(* PLC project PLC Garden Controller, CODESYS CODESYS V3.5 SP16, author Toni Kucic *)
(* stored: creationDateTime 2021-03-29T22:16:35.9497507, version 1.0, modificationDateTime 2021-03-29T21:41:22.9745241, organization TK Automation *)
(* Automated gardening at its best. This is a portfolio project that features a simulator and a controller of four gardens holding 25 flowers/plants each. Each garden has a watering platform system moved by servo motors. In this project the user can learn how to control servo motors, optimize instruction/path algorithms and generally learn how to program PLCs. *)

TYPE Flower_typ : STRUCT
  x : INT;  (* X position of the flower cell in the HMI *)
  y : INT;  (* Y position of the flower cell in the HMI *)
  alpha : BYTE := 255;  (* Alpha channel *)
  red : BYTE := 2;  (* Red color channel *)
  green : BYTE := 253;  (* Green color channel *)
  blue : BYTE := 0;  (* Blue color channel *)
  color : DWORD;  (* Color variable to be used in the graphics *)
  hum : REAL := 100;  (* Humidity of the flower cell *)
  alive : BOOL := TRUE;  (* Flower is alive *)
END_STRUCT;
END_TYPE

TYPE Platform_typ : STRUCT
  x : INT;  (* Position from starting point on X axis *)
  y : INT;  (* Position from starting point on Y axis *)
  OpenValveCmd : BOOL;  (* Opens the water container valve *)
END_STRUCT;
END_TYPE

TYPE HMI_Cmds_typ : STRUCT
  CtrlOn : BOOL := TRUE;  (* Control is activated *)
  UpCmd : BOOL;  (* Command for platform UP *)
  DownCmd : BOOL;  (* Command for platform DOWN *)
  LeftCmd : BOOL;  (* Command for platform LEFT *)
  RightCmd : BOOL;  (* Command for platform RIGHT *)
  LeftUpCmd : BOOL;  (* Command for platform LEFT AND UP *)
  RightUpCmd : BOOL;  (* Command for platform RIGHT AND UP *)
  LeftDownCmd : BOOL;  (* Command for platform LEFT AND DOWN *)
  RightDownCmd : BOOL;  (* Command for platform RIGHT AND DOWN *)
  OpenWaterValve : BOOL;  (* Command to open the water valve *)
END_STRUCT;
END_TYPE

FUNCTION BYTES_TO_DWORD : DWORD
  VAR_INPUT
    B0 : BYTE;  (* Least significant byte *)
    B1 : BYTE;  (* Byte two *)
    B2 : BYTE;  (* Byte three *)
    B3 : BYTE;  (* Highest significant byte *)
  END_VAR

            BYTES_TO_DWORD.0 := B0.0;
BYTES_TO_DWORD.1 := B0.1;
BYTES_TO_DWORD.2 := B0.2;
BYTES_TO_DWORD.3 := B0.3;
BYTES_TO_DWORD.4 := B0.4;
BYTES_TO_DWORD.5 := B0.5;
BYTES_TO_DWORD.6 := B0.6;
BYTES_TO_DWORD.7 := B0.7;

BYTES_TO_DWORD.8 := B1.0;
BYTES_TO_DWORD.9 := B1.1;
BYTES_TO_DWORD.10 := B1.2;
BYTES_TO_DWORD.11 := B1.3;
BYTES_TO_DWORD.12 := B1.4;
BYTES_TO_DWORD.13 := B1.5;
BYTES_TO_DWORD.14 := B1.6;
BYTES_TO_DWORD.15 := B1.7;

BYTES_TO_DWORD.16 := B2.0;
BYTES_TO_DWORD.17 := B2.1;
BYTES_TO_DWORD.18 := B2.2;
BYTES_TO_DWORD.19 := B2.3;
BYTES_TO_DWORD.20 := B2.4;
BYTES_TO_DWORD.21 := B2.5;
BYTES_TO_DWORD.22 := B2.6;
BYTES_TO_DWORD.23 := B2.7;

BYTES_TO_DWORD.24 := B3.0;
BYTES_TO_DWORD.25 := B3.1;
BYTES_TO_DWORD.26 := B3.2;
BYTES_TO_DWORD.27 := B3.3;
BYTES_TO_DWORD.28 := B3.4;
BYTES_TO_DWORD.29 := B3.5;
BYTES_TO_DWORD.30 := B3.6;
BYTES_TO_DWORD.31 := B3.7;
RETURN;
          
END_FUNCTION

FUNCTION_BLOCK ClockPulse
  VAR_INPUT
    f : TIME := TIME#500ms;  (* Oscillate once per f *)
  END_VAR
  VAR_OUTPUT
    pulse : BOOL;  (* Pulse for use. One cycle *)
  END_VAR
  VAR
    edge : R_TRIG;
    clock : BLINK;
  END_VAR

            clock(ENABLE:=TRUE, TIMELOW:=f, TIMEHIGH:=f);
edge(CLK:=clock.OUT);
pulse := edge.Q;
          
END_FUNCTION_BLOCK

FUNCTION checkOverlapRectangle : BOOL
  VAR_INPUT
    R1_X : INT;  (* Rectangle 1 x position *)
    R1_Y : INT;  (* Rectangle 1 y position *)
    R1_W : INT;  (* Rectangle 1 width *)
    R1_H : INT;  (* Rectangle 1 height *)
    R2_X : INT;  (* Rectangle 2 x position *)
    R2_Y : INT;  (* Rectangle 2 y position *)
    R2_W : INT;  (* Rectangle 2 width *)
    R2_H : INT;  (* Rectangle 2 height *)
  END_VAR

            (*Calculate if these two rectangles are overlapping*)
IF R1_X < (R2_X + R2_W) AND
   (R1_X + R1_W) > R2_X AND
   R1_Y < (R2_Y + R2_H) AND
  (R1_H + R1_Y) > R2_Y THEN
   checkOverlapRectangle := TRUE;
ELSE
	checkOverlapRectangle := FALSE;
END_IF
          
END_FUNCTION

PROGRAM simu
  VAR
    clock : ClockPulse;  (* Clock pulse for the program *)
    i : UINT;  (* Iterator variable *)
    vG1PlantsAlive : UINT;  (* Number of plants alive in garden 1 *)
    vG2PlantsAlive : UINT;  (* Number of plants alive in garden 2 *)
    vG3PlantsAlive : UINT;  (* Number of plants alive in garden 3 *)
    vG4PlantsAlive : UINT;  (* Number of plants alive in garden 4 *)
    vGarden1 : ARRAY[0..24] OF Flower_typ := [(x := 42, y := 42), (x := 122, y := 42), (x := 202, y := 42), (x := 282, y := 42), (x := 362, y := 42), (x := 42, y := 122), (x := 122, y := 122), (x := 202, y := 122), (x := 282, y := 122), (x := 362, y := 122), (x := 42, y := 202), (x := 122, y := 202), (x := 202, y := 202), (x := 282, y := 202), (x := 362, y := 202), (x := 42, y := 282), (x := 122, y := 282), (x := 202, y := 282), (x := 282, y := 282), (x := 362, y := 282), (x := 42, y := 362), (x := 122, y := 362), (x := 202, y := 362), (x := 282, y := 362), (x := 362, y := 362)];  (* Locations of plant cells in the HMI for the garden 1. Not to be mistaken with servo offset *)
    vGarden2 : ARRAY[0..24] OF Flower_typ := [(x := 642, y := 42), (x := 722, y := 42), (x := 802, y := 42), (x := 882, y := 42), (x := 962, y := 42), (x := 642, y := 122), (x := 722, y := 122), (x := 802, y := 122), (x := 882, y := 122), (x := 962, y := 122), (x := 642, y := 202), (x := 722, y := 202), (x := 802, y := 202), (x := 882, y := 202), (x := 962, y := 202), (x := 642, y := 282), (x := 722, y := 282), (x := 802, y := 282), (x := 882, y := 282), (x := 962, y := 282), (x := 642, y := 362), (x := 722, y := 362), (x := 802, y := 362), (x := 882, y := 362), (x := 962, y := 362)];  (* Locations of plant cells in the HMI for the garden 2. Not to be mistaken with servo offset *)
    vGarden3 : ARRAY[0..24] OF Flower_typ := [(x := 42, y := 642), (x := 122, y := 642), (x := 202, y := 642), (x := 282, y := 642), (x := 362, y := 642), (x := 42, y := 722), (x := 122, y := 722), (x := 202, y := 722), (x := 282, y := 722), (x := 362, y := 722), (x := 42, y := 802), (x := 122, y := 802), (x := 202, y := 802), (x := 282, y := 802), (x := 362, y := 802), (x := 42, y := 882), (x := 122, y := 882), (x := 202, y := 882), (x := 282, y := 882), (x := 362, y := 882), (x := 42, y := 962), (x := 122, y := 962), (x := 202, y := 962), (x := 282, y := 962), (x := 362, y := 962)];  (* Locations of plant cells in the HMI for the garden 3. Not to be mistaken with servo offset *)
    vGarden4 : ARRAY[0..24] OF Flower_typ := [(x := 642, y := 642), (x := 722, y := 642), (x := 802, y := 642), (x := 882, y := 642), (x := 962, y := 642), (x := 642, y := 722), (x := 722, y := 722), (x := 802, y := 722), (x := 882, y := 722), (x := 962, y := 722), (x := 642, y := 802), (x := 722, y := 802), (x := 802, y := 802), (x := 882, y := 802), (x := 962, y := 802), (x := 642, y := 882), (x := 722, y := 882), (x := 802, y := 882), (x := 882, y := 882), (x := 962, y := 882), (x := 642, y := 962), (x := 722, y := 962), (x := 802, y := 962), (x := 882, y := 962), (x := 962, y := 962)];  (* Locations of plant cells in the HMI for the garden 4. Not to be mistaken with servo offset *)
    vGarden1Platform : Platform_typ;  (* Platform 1 properties like x,y, water valve open etc *)
    vGarden2Platform : Platform_typ;  (* Platform 2 properties like x,y, water valve open etc *)
    vGarden3Platform : Platform_typ;  (* Platform 3 properties like x,y, water valve open etc *)
    vGarden4Platform : Platform_typ;  (* Platform 4 properties like x,y, water valve open etc *)
  END_VAR

                    (* SIMULATOR FUNCTIONAL DESCRIPTION
FLOWERS SIMULATION:
- there are 25 flowers in each garden
- each flower consumes humidity for life, this is represented as a number, this draw is constant
- each flower, if it has no humidity, it start decaying, decaying is represented with color
if color is red, the flower dies, if its green or yellow it is still alive
- if the flower gets too much water (>200%) this has same effect as it being too dry so the 
platform controller must maintain a proper level of humidity.
- there are no humidity sensors deployed to the gIO structure but if the user wants to, it is very easy

PLATFORM SIMULATION:
- platforms consist out of one Y Axis servo and two X axis servos
- X axis servos are electrically connected so they move as one for simplicity
- each servo motor is reporting its offset from the beggining of the servo
- for simplicity, each servo starts at 0 offset. If necessary, these starting points can be initialized
- commands CW increase the axis while CCW decrease the axis
- servo motors are identical but they are  flipped horizontally or verticaly, depending on the garden
but they always follow CW and CCW commands respectively
- upon command the open water valve releases the onboard stored water. For simplicity, the platform has 
unlimited supply of water

PLATFORM/FLOWER INTERACTION SIMULATION:
- if the nozzle (not the whole platform) of the platform is above a flower cell (80x80 pixels)
and the water valve is open, the flowers humidity increases
- the flower cells are divided by 1 px width and the nozzle is 10px wide so it is possible to
water multiple cells at once

COUNTING OF ALIVE FLOWERS:
- for each garden a counting of alive plants is done and it is displayed in the HMI*)

clock(f:=T#20MS);

(*Run the garden simulators*)
SIMULATE_GARDEN1();
SIMULATE_GARDEN2();
SIMULATE_GARDEN3();
SIMULATE_GARDEN4();
                  

ACTION SIMULATE_GARDEN1:
                        (*COLOR : 16# XX XX XX XX*)
(*            A  R  G  B *)
vG1PlantsAlive := 0;
FOR i:=0 TO 24 DO
	(*Simulate the humidity of one flower cell*)
	(*If not being watered, it slowly looses humidity*)
	vGarden1[i].hum := MAX(0, vGarden1[i].hum - 0.07 * BOOL_TO_REAL(clock.pulse));
	
	(*If the watering platform is above the cell, water valve is open and tank has water, increase the humidity*)
	IF checkOverlapRectangle(R1_X:=vGarden1[i].x, R1_Y:=vGarden1[i].y, R1_W:=80, R1_H:=80,
							R2_X:=406 + vGarden1Platform.x + 45, R2_Y:=361 + vGarden1Platform.y + 45, R2_W:=10, R2_H:=10) AND vGarden1Platform.OpenValveCmd THEN
		vGarden1[i].hum := vGarden1[i].hum + 4 * BOOL_TO_REAL(clock.pulse);
	END_IF
	
	(*Simulate flowers response to the humidity of the cell*)
	(*Flag if the plant is alive*)
	vGarden1[i].alive := NOT (vGarden1[i].red >= 254 AND vGarden1[i].green < 100);
	IF vGarden1[i].hum <= 0 OR vGarden1[i].hum >= 200 THEN
		(*Flower starts decaying if not enough or too much humiditiy*)
		(*Change color towards red*)
		vGarden1[i].red := vGarden1[i].red + 1 * BOOL_TO_BYTE(clock.pulse);
		vGarden1[i].green := vGarden1[i].green - 1 * BOOL_TO_BYTE(clock.pulse AND vGarden1[i].red > 253);
	ELSE
		IF vGarden1[i].alive THEN
			(*Flower gets better much faster than it dies*)
			(*Change color towards green*)
			vGarden1[i].green := vGarden1[i].green + 1 * BOOL_TO_BYTE(clock.pulse);
			vGarden1[i].red := vGarden1[i].red - 1 * BOOL_TO_BYTE(clock.pulse AND vGarden1[i].green > 253);
		(*ELSE It is dead for good*)
			
		END_IF
	END_IF
	vGarden1[i].red := LIMIT(1, vGarden1[i].red, 254);
	vGarden1[i].green := LIMIT(1, vGarden1[i].green, 254);
	
	(*Combine the channel bytes into dword color*)
	vGarden1[i].color := BYTES_TO_DWORD(B0 := vGarden1[i].blue,B1 := vGarden1[i].green,
										B2 := vGarden1[i].red, B3 := vGarden1[i].alpha);
										
	(*Count how many plants are alive*)
	vG1PlantsAlive := vG1PlantsAlive + BOOL_TO_UINT(vGarden1[i].alive);
END_FOR

(*Servo motors*)
(*Move on X*)
IF gIO.Garden1_ServoX_CCW THEN
	vGarden1Platform.x := vGarden1Platform.x + 1;
ELSIF gIO.Garden1_ServoX_CW THEN
	vGarden1Platform.x := vGarden1Platform.x - 1;
END_IF
(*Limit the platforms movement on x axis*)
vGarden1Platform.x := LIMIT(-404, vGarden1Platform.x, 0);
(*Move on Y*)
IF gIO.Garden1_ServoY_CCW THEN
	vGarden1Platform.y := vGarden1Platform.y + 1;
ELSIF gIO.Garden1_ServoY_CW THEN
	vGarden1Platform.y := vGarden1Platform.y - 1;
END_IF
(*Limit the platforms movement on y axis*)
vGarden1Platform.y := LIMIT(-320, vGarden1Platform.y, 0);

(*Report the position of the platform*)
gIO.Garden1_ServoX_Offset := ABS(vGarden1Platform.x);
gIO.Garden1_ServoY_Offset := ABS(vGarden1Platform.y);

(*Control the water valve*)
vGarden1Platform.OpenValveCmd := gIO.Garden1_WaterTankOpenCmd;
                      
END_ACTION

ACTION SIMULATE_GARDEN2:
                        (*COLOR : 16# XX XX XX XX*)
(*            A  R  G  B *)
vG2PlantsAlive := 0;
FOR i:=0 TO 24 DO
	(*Simulate the humidity of one flower cell*)
	(*If not being watered, it slowly looses humidity*)
	vGarden2[i].hum := MAX(0, vGarden2[i].hum - 0.07 * BOOL_TO_REAL(clock.pulse));
	
	(*If the watering platform is above the cell, water valve is open and tank has water, increase the humidity*)
	IF checkOverlapRectangle(R1_X:=vGarden2[i].x, R1_Y:=vGarden2[i].y, R1_W:=80, R1_H:=80,
							R2_X:=594 + vGarden2Platform.x + 45, R2_Y:=361 + vGarden2Platform.y + 45, R2_W:=10, R2_H:=10) AND vGarden2Platform.OpenValveCmd THEN
		vGarden2[i].hum := vGarden2[i].hum + 4 * BOOL_TO_REAL(clock.pulse);
	END_IF
	
	(*Simulate flowers response to the humidity of the cell*)
	(*Flag if the plant is alive*)
	vGarden2[i].alive := NOT (vGarden2[i].red >= 254 AND vGarden2[i].green < 100);
	IF vGarden2[i].hum <= 0 OR vGarden2[i].hum >= 200 THEN
		(*Flower starts decaying if not enough or too much humiditiy*)
		(*Change color towards red*)
		vGarden2[i].red := vGarden2[i].red + 1 * BOOL_TO_BYTE(clock.pulse);
		vGarden2[i].green := vGarden2[i].green - 1 * BOOL_TO_BYTE(clock.pulse AND vGarden2[i].red > 253);
	ELSE
		IF vGarden2[i].alive THEN
			(*Flower gets better much faster than it dies*)
			(*Change color towards green*)
			vGarden2[i].green := vGarden2[i].green + 1 * BOOL_TO_BYTE(clock.pulse);
			vGarden2[i].red := vGarden2[i].red - 1 * BOOL_TO_BYTE(clock.pulse AND vGarden2[i].green > 253);
		(*ELSE It is dead for good*)
			
		END_IF
	END_IF
	vGarden2[i].red := LIMIT(1, vGarden2[i].red, 254);
	vGarden2[i].green := LIMIT(1, vGarden2[i].green, 254);
	
	(*Combine the channel bytes into dword color*)
	vGarden2[i].color := BYTES_TO_DWORD(B0 := vGarden2[i].blue,B1 := vGarden2[i].green,
										B2 := vGarden2[i].red, B3 := vGarden2[i].alpha);
										
	(*Count how many plants are alive*)
	vG2PlantsAlive := vG2PlantsAlive + BOOL_TO_UINT(vGarden2[i].alive);
END_FOR

(*Servo motors*)
(*Move on X*)
IF gIO.Garden2_ServoX_CCW THEN
	vGarden2Platform.x := vGarden2Platform.x - 1;
ELSIF gIO.Garden2_ServoX_CW THEN
	vGarden2Platform.x := vGarden2Platform.x + 1;
END_IF
(*Limit the platforms movement on x axis*)
vGarden2Platform.x := LIMIT(0, vGarden2Platform.x, 404);
(*Move on Y*)
IF gIO.Garden2_ServoY_CCW THEN
	vGarden2Platform.y := vGarden2Platform.y + 1;
ELSIF gIO.Garden2_ServoY_CW THEN
	vGarden2Platform.y := vGarden2Platform.y - 1;
END_IF
(*Limit the platforms movement on y axis*)
vGarden2Platform.y := LIMIT(-320, vGarden2Platform.y, 0);

(*Report the position of the platform*)
gIO.Garden2_ServoX_Offset := ABS(vGarden2Platform.x);
gIO.Garden2_ServoY_Offset := ABS(vGarden2Platform.y);

(*Control the water valve*)
vGarden2Platform.OpenValveCmd := gIO.Garden2_WaterTankOpenCmd;
                      
END_ACTION

ACTION SIMULATE_GARDEN3:
                        (*COLOR : 16# XX XX XX XX*)
(*            A  R  G  B *)
vG3PlantsAlive := 0;
FOR i:=0 TO 24 DO
	(*Simulate the humidity of one flower cell*)
	(*If not being watered, it slowly looses humidity*)
	vGarden3[i].hum := MAX(0, vGarden3[i].hum - 0.07 * BOOL_TO_REAL(clock.pulse));
	
	(*If the watering platform is above the cell, water valve is open and tank has water, increase the humidity*)
	IF checkOverlapRectangle(R1_X:=vGarden3[i].x, R1_Y:=vGarden3[i].y, R1_W:=80, R1_H:=80,
							R2_X:=401 + vGarden3Platform.x + 45, R2_Y:=640 + vGarden3Platform.y + 45, R2_W:=10, R2_H:=10) AND vGarden3Platform.OpenValveCmd THEN
		vGarden3[i].hum := vGarden3[i].hum + 4 * BOOL_TO_REAL(clock.pulse);
	END_IF
	
	(*Simulate flowers response to the humidity of the cell*)
	(*Flag if the plant is alive*)
	vGarden3[i].alive := NOT (vGarden3[i].red >= 254 AND vGarden3[i].green < 100);
	IF vGarden3[i].hum <= 0 OR vGarden3[i].hum >= 200 THEN
		(*Flower starts decaying if not enough or too much humiditiy*)
		(*Change color towards red*)
		vGarden3[i].red := vGarden3[i].red + 1 * BOOL_TO_BYTE(clock.pulse);
		vGarden3[i].green := vGarden3[i].green - 1 * BOOL_TO_BYTE(clock.pulse AND vGarden3[i].red > 253);
	ELSE
		IF vGarden3[i].alive THEN
			(*Flower gets better much faster than it dies*)
			(*Change color towards green*)
			vGarden3[i].green := vGarden3[i].green + 1 * BOOL_TO_BYTE(clock.pulse);
			vGarden3[i].red := vGarden3[i].red - 1 * BOOL_TO_BYTE(clock.pulse AND vGarden3[i].green > 253);
		(*ELSE It is dead for good*)
			
		END_IF
	END_IF
	vGarden3[i].red := LIMIT(1, vGarden3[i].red, 254);
	vGarden3[i].green := LIMIT(1, vGarden3[i].green, 254);
	
	(*Combine the channel bytes into dword color*)
	vGarden3[i].color := BYTES_TO_DWORD(B0 := vGarden3[i].blue,B1 := vGarden3[i].green,
										B2 := vGarden3[i].red, B3 := vGarden3[i].alpha);
										
	(*Count how many plants are alive*)
	vG3PlantsAlive := vG3PlantsAlive + BOOL_TO_UINT(vGarden3[i].alive);
END_FOR

(*Servo motors*)
(*Move on X*)
IF gIO.Garden3_ServoX_CCW THEN
	vGarden3Platform.x := vGarden3Platform.x + 1;
ELSIF gIO.Garden3_ServoX_CW THEN
	vGarden3Platform.x := vGarden3Platform.x - 1;
END_IF
(*Limit the platforms movement on x axis*)
vGarden3Platform.x := LIMIT(-404, vGarden3Platform.x, 0);
(*Move on Y*)
IF gIO.Garden3_ServoY_CCW THEN
	vGarden3Platform.y := vGarden3Platform.y - 1;
ELSIF gIO.Garden3_ServoY_CW THEN
	vGarden3Platform.y := vGarden3Platform.y + 1;
END_IF
(*Limit the platforms movement on y axis*)
vGarden3Platform.y := LIMIT(0, vGarden3Platform.y, 320);

(*Report the position of the platform*)
gIO.Garden3_ServoX_Offset := ABS(vGarden3Platform.x);
gIO.Garden3_ServoY_Offset := ABS(vGarden3Platform.y);

(*Control the water valve*)
vGarden3Platform.OpenValveCmd := gIO.Garden3_WaterTankOpenCmd;
                      
END_ACTION

ACTION SIMULATE_GARDEN4:
                        (*COLOR : 16# XX XX XX XX*)
(*            A  R  G  B *)
vG4PlantsAlive := 0;
FOR i:=0 TO 24 DO
	(*Simulate the humidity of one flower cell*)
	(*If not being watered, it slowly looses humidity*)
	vGarden4[i].hum := MAX(0, vGarden4[i].hum - 0.07 * BOOL_TO_REAL(clock.pulse));
	
	(*If the watering platform is above the cell, water valve is open and tank has water, increase the humidity*)
	IF checkOverlapRectangle(R1_X:=vGarden4[i].x, R1_Y:=vGarden4[i].y, R1_W:=80, R1_H:=80,
							R2_X:=600 + vGarden4Platform.x + 45, R2_Y:=642 + vGarden4Platform.y + 45, R2_W:=10, R2_H:=10) AND vGarden4Platform.OpenValveCmd THEN
		vGarden4[i].hum := vGarden4[i].hum + 4 * BOOL_TO_REAL(clock.pulse);
	END_IF
	
	(*Simulate flowers response to the humidity of the cell*)
	(*Flag if the plant is alive*)
	vGarden4[i].alive := NOT (vGarden4[i].red >= 254 AND vGarden4[i].green < 100);
	IF vGarden4[i].hum <= 0 OR vGarden4[i].hum >= 200 THEN
		(*Flower starts decaying if not enough or too much humiditiy*)
		(*Change color towards red*)
		vGarden4[i].red := vGarden4[i].red + 1 * BOOL_TO_BYTE(clock.pulse);
		vGarden4[i].green := vGarden4[i].green - 1 * BOOL_TO_BYTE(clock.pulse AND vGarden4[i].red > 253);
	ELSE
		IF vGarden4[i].alive THEN
			(*Flower gets better much faster than it dies*)
			(*Change color towards green*)
			vGarden4[i].green := vGarden4[i].green + 1 * BOOL_TO_BYTE(clock.pulse);
			vGarden4[i].red := vGarden4[i].red - 1 * BOOL_TO_BYTE(clock.pulse AND vGarden4[i].green > 253);
		(*ELSE It is dead for good*)
			
		END_IF
	END_IF
	vGarden4[i].red := LIMIT(1, vGarden4[i].red, 254);
	vGarden4[i].green := LIMIT(1, vGarden4[i].green, 254);
	
	(*Combine the channel bytes into dword color*)
	vGarden4[i].color := BYTES_TO_DWORD(B0 := vGarden4[i].blue,B1 := vGarden4[i].green,
										B2 := vGarden4[i].red, B3 := vGarden4[i].alpha);
										
	(*Count how many plants are alive*)
	vG4PlantsAlive := vG4PlantsAlive + BOOL_TO_UINT(vGarden4[i].alive);
END_FOR

(*Servo motors*)
(*Move on X*)
IF gIO.Garden4_ServoX_CCW THEN
	vGarden4Platform.x := vGarden4Platform.x - 1;
ELSIF gIO.Garden4_ServoX_CW THEN
	vGarden4Platform.x := vGarden4Platform.x + 1;
END_IF
(*Limit the platforms movement on x axis*)
vGarden4Platform.x := LIMIT(0, vGarden4Platform.x, 404);
(*Move on Y*)
IF gIO.Garden4_ServoY_CCW THEN
	vGarden4Platform.y := vGarden4Platform.y - 1;
ELSIF gIO.Garden4_ServoY_CW THEN
	vGarden4Platform.y := vGarden4Platform.y + 1;
END_IF
(*Limit the platforms movement on y axis*)
vGarden4Platform.y := LIMIT(0, vGarden4Platform.y, 320);

(*Report the position of the platform*)
gIO.Garden4_ServoX_Offset := ABS(vGarden4Platform.x);
gIO.Garden4_ServoY_Offset := ABS(vGarden4Platform.y);

(*Control the water valve*)
vGarden4Platform.OpenValveCmd := gIO.Garden4_WaterTankOpenCmd;
                      
END_ACTION
END_PROGRAM

PROGRAM main
  VAR
    vG1Platform_Instructions : ARRAY[0..24, 0..1] OF INT := [365, 320, 285, 320, 205, 320, 125, 320, 45, 320, 45, 240, 125, 240, 205, 240, 285, 240, 365, 240, 365, 160, 285, 160, 205, 160, 125, 160, 45, 160, 45, 80, 125, 80, 205, 80, 285, 80, 365, 80, 365, 0, 285, 0, 205, 0, 125, 0, 45, 0];  (* Instructions for platform servos in garden 1 *)
    vG2Platform_Instructions : ARRAY[0..24, 0..1] OF INT := [50, 320, 50, 240, 50, 160, 50, 80, 50, 0, 130, 0, 130, 80, 130, 160, 130, 240, 130, 320, 210, 320, 210, 240, 210, 160, 210, 80, 210, 0, 290, 0, 290, 80, 290, 160, 290, 240, 290, 320, 370, 320, 370, 240, 370, 160, 370, 80, 370, 0];  (* Instructions for platform servos in garden 2 *)
    vG3Platform_Instructions : ARRAY[0..24, 0..1] OF INT := [358, 0, 278, 0, 358, 80, 358, 160, 278, 80, 198, 0, 118, 0, 198, 80, 278, 160, 358, 240, 358, 320, 278, 240, 198, 160, 118, 80, 38, 0, 38, 80, 118, 160, 198, 240, 278, 320, 198, 320, 118, 240, 38, 160, 38, 240, 118, 320, 38, 320];  (* Instructions for platform servos in garden 3 *)
    vG4Platform_Instructions : ARRAY[0..24, 0..1] OF INT := [200, 160, 120, 160, 120, 240, 200, 240, 280, 240, 280, 160, 280, 80, 200, 80, 120, 80, 40, 80, 40, 160, 40, 240, 40, 320, 120, 320, 200, 320, 280, 320, 360, 320, 360, 240, 360, 160, 360, 80, 360, 0, 280, 0, 200, 0, 120, 0, 40, 0];  (* Instructions for platform servos in garden 4 *)
    garden1AutoWater : AutomaticFlowerWatering;  (* Automatic watering logic: Left to right in a smart way *)
    garden2AutoWater : AutomaticFlowerWatering;  (* Automatic watering logic: Going top to bottom in a smart way *)
    garden3AutoWater : AutomaticFlowerWatering;  (* Automatic watering logic: Going side ways from the top to bottom *)
    garden4AutoWater : AutomaticFlowerWatering;  (* Automatic watering logic: Goign from the middle out *)
  END_VAR

                    (*FUNCTIONAL DESCRIPTION:
- there are four gardens holding 25 flowers each
- the flowers need to be watered on a regular basis in order to keep their humidity in correct levels
- correct humidity is 0 > x < 200 %, if the humidity is not in those limits, the flower starts dying
- the watering is done by means of a watering platform, moved by x a y servos
- the job of this program is to move the platform of each garden and water the plants in an optimized way
- program should strive to keep all plants alive (easier said than done)
- the platforms move quite slowly as the water tank might spill so it is a given that 25 flower can be 
watered in 25 seconds
- on top of each platform there is a water tank with a valve that can be open remotely by the main program
- the program also needs to implement manual control from the HMI with the prepared variables in gIO structure
*)
CONTROL_GARDEN1();
CONTROL_GARDEN2();
CONTROL_GARDEN3();
CONTROL_GARDEN4();

                  

ACTION CONTROL_GARDEN1:
                        IF gIO.Garden1_HMI.CtrlOn THEN
	(*HMI Control*)
	gIO.Garden1_ServoX_CW := gIO.Garden1_HMI.LeftCmd OR gIO.Garden1_HMI.LeftDownCmd OR gIO.Garden1_HMI.LeftUpCmd;
	gIO.Garden1_ServoX_CCW := gIO.Garden1_HMI.RightCmd OR gIO.Garden1_HMI.RightDownCmd OR gIO.Garden1_HMI.RightUpCmd;
	
	gIO.Garden1_ServoY_CW := gIO.Garden1_HMI.UpCmd OR gIO.Garden1_HMI.LeftUpCmd OR gIO.Garden1_HMI.RightUpCmd;
	gIO.Garden1_ServoY_CCW := gIO.Garden1_HMI.DownCmd OR gIO.Garden1_HMI.LeftDownCmd OR gIO.Garden1_HMI.RightDownCmd;
	
	gIO.Garden1_WaterTankOpenCmd := gIO.Garden1_HMI.OpenWaterValve;
ELSE
	(*Automatic control*)
	garden1AutoWater(instructions:=vG1Platform_Instructions,
		xAxis := gIO.Garden1_ServoX_Offset,
		yAxis := gIO.Garden1_ServoY_Offset,
		servoX_CW => gIO.Garden1_ServoX_CW,
		servoX_CCW => gIO.Garden1_ServoX_CCW,
		servoY_CW => gIO.Garden1_ServoY_CW,
		servoY_CCW => gIO.Garden1_ServoY_CCW,
		waterTankOpenCmd => gIO.Garden1_WaterTankOpenCmd);
END_IF
                      
END_ACTION

ACTION CONTROL_GARDEN2:
                        IF gIO.Garden2_HMI.CtrlOn THEN
	(*HMI Control*)
	(*X servos are flipped on this garden*)
	gIO.Garden2_ServoX_CCW := gIO.Garden2_HMI.LeftCmd OR gIO.Garden2_HMI.LeftDownCmd OR gIO.Garden2_HMI.LeftUpCmd;
	gIO.Garden2_ServoX_CW := gIO.Garden2_HMI.RightCmd OR gIO.Garden2_HMI.RightDownCmd OR gIO.Garden2_HMI.RightUpCmd;
	
	gIO.Garden2_ServoY_CW := gIO.Garden2_HMI.UpCmd OR gIO.Garden2_HMI.LeftUpCmd OR gIO.Garden2_HMI.RightUpCmd;
	gIO.Garden2_ServoY_CCW := gIO.Garden2_HMI.DownCmd OR gIO.Garden2_HMI.LeftDownCmd OR gIO.Garden2_HMI.RightDownCmd;
	
	gIO.Garden2_WaterTankOpenCmd := gIO.Garden2_HMI.OpenWaterValve;
ELSE
	(*Automatic control*)
	garden2AutoWater(instructions:=vG2Platform_Instructions,
		xAxis := gIO.Garden2_ServoX_Offset,
		yAxis := gIO.Garden2_ServoY_Offset,
		servoX_CW => gIO.Garden2_ServoX_CW,
		servoX_CCW => gIO.Garden2_ServoX_CCW,
		servoY_CW => gIO.Garden2_ServoY_CW,
		servoY_CCW => gIO.Garden2_ServoY_CCW,
		waterTankOpenCmd => gIO.Garden2_WaterTankOpenCmd);
END_IF
                      
END_ACTION

ACTION CONTROL_GARDEN3:
                        IF gIO.Garden3_HMI.CtrlOn THEN
	(*HMI Control*)
	gIO.Garden3_ServoX_CW := gIO.Garden3_HMI.LeftCmd OR gIO.Garden3_HMI.LeftDownCmd OR gIO.Garden3_HMI.LeftUpCmd;
	gIO.Garden3_ServoX_CCW := gIO.Garden3_HMI.RightCmd OR gIO.Garden3_HMI.RightDownCmd OR gIO.Garden3_HMI.RightUpCmd;
	
	gIO.Garden3_ServoY_CCW := gIO.Garden3_HMI.UpCmd OR gIO.Garden3_HMI.LeftUpCmd OR gIO.Garden3_HMI.RightUpCmd;
	gIO.Garden3_ServoY_CW := gIO.Garden3_HMI.DownCmd OR gIO.Garden3_HMI.LeftDownCmd OR gIO.Garden3_HMI.RightDownCmd;
	
	gIO.Garden3_WaterTankOpenCmd := gIO.Garden3_HMI.OpenWaterValve;
ELSE
	(*Automatic control*)
	garden3AutoWater(instructions:=vG3Platform_Instructions,
		xAxis := gIO.Garden3_ServoX_Offset,
		yAxis := gIO.Garden3_ServoY_Offset,
		servoX_CW => gIO.Garden3_ServoX_CW,
		servoX_CCW => gIO.Garden3_ServoX_CCW,
		servoY_CW => gIO.Garden3_ServoY_CW,
		servoY_CCW => gIO.Garden3_ServoY_CCW,
		waterTankOpenCmd => gIO.Garden3_WaterTankOpenCmd);
END_IF
                      
END_ACTION

ACTION CONTROL_GARDEN4:
                        IF gIO.Garden4_HMI.CtrlOn THEN
	(*HMI Control*)
	gIO.Garden4_ServoX_CCW := gIO.Garden4_HMI.LeftCmd OR gIO.Garden4_HMI.LeftDownCmd OR gIO.Garden4_HMI.LeftUpCmd;
	gIO.Garden4_ServoX_CW := gIO.Garden4_HMI.RightCmd OR gIO.Garden4_HMI.RightDownCmd OR gIO.Garden4_HMI.RightUpCmd;
	
	gIO.Garden4_ServoY_CCW := gIO.Garden4_HMI.UpCmd OR gIO.Garden4_HMI.LeftUpCmd OR gIO.Garden4_HMI.RightUpCmd;
	gIO.Garden4_ServoY_CW := gIO.Garden4_HMI.DownCmd OR gIO.Garden4_HMI.LeftDownCmd OR gIO.Garden4_HMI.RightDownCmd;
	
	gIO.Garden4_WaterTankOpenCmd := gIO.Garden4_HMI.OpenWaterValve;
ELSE
	(*Automatic control*)
	garden4AutoWater(instructions:=vG4Platform_Instructions,
		xAxis := gIO.Garden4_ServoX_Offset,
		yAxis := gIO.Garden4_ServoY_Offset,
		servoX_CW => gIO.Garden4_ServoX_CW,
		servoX_CCW => gIO.Garden4_ServoX_CCW,
		servoY_CW => gIO.Garden4_ServoY_CW,
		servoY_CCW => gIO.Garden4_ServoY_CCW,
		waterTankOpenCmd => gIO.Garden4_WaterTankOpenCmd);
END_IF
                      
END_ACTION
END_PROGRAM

FUNCTION_BLOCK AutomaticFlowerWatering
  VAR_INPUT
    instructions : ARRAY[0..24, 0..1] OF INT;  (* Instructions to follow *)
    xAxis : INT;  (* Actual position of the X axis servo *)
    yAxis : INT;  (* Actual position of the Y axis servo *)
  END_VAR
  VAR_OUTPUT
    servoX_CW : BOOL;  (* Command to turn X axis servo clock wise *)
    servoX_CCW : BOOL;  (* Command to turn X axis servo counter clock wise *)
    servoY_CW : BOOL;  (* Command to turn Y axis servo clock wise *)
    servoY_CCW : BOOL;  (* Command to turn Y axis servo counter clock wise *)
    waterTankOpenCmd : BOOL;  (* Command to the platform to open the water valve *)
  END_VAR
  VAR
    i : UINT;  (* Iterator variable *)
    vXAxisCmd : INT;  (* Next X axis target *)
    vYAxisCmd : INT;  (* Next Y axis target *)
    vPlatformAtTarget : BOOL;  (* Flag for reaching the target *)
    WateringTimer : TON;  (* Timer for controlling the valve being open *)
  END_VAR

                    (* Parse the instruction to get new x and y targets *)
vXAxisCmd := instructions[i,0];
vYAxisCmd := instructions[i,1];
	
(*Check if the platform is at the target*)
vPlatformAtTarget := xAxis = vXAxisCmd AND yAxis = vYAxisCmd;

IF vPlatformAtTarget THEN
	(*Start watering for 1 second*)
	WateringTimer(IN:=TRUE, PT:=T#1S);
	waterTankOpenCmd := TRUE;
	
	(*If watering is finished, close valve and go to next flower*)
	IF WateringTimer.Q THEN
		WateringTimer(IN := FALSE);
		waterTankOpenCmd:= FALSE;
		i:= i + 1;
	END_IF
END_IF

(*If we traversed all instructions, go to first instruction*)
IF i = 25 THEN
	i := 0;
END_IF

(* Actual motor movement algorithm *)
IF vXAxisCmd > xAxis THEN
	servoX_CCW := FALSE;
	servoX_CW := TRUE;
ELSIF vXAxisCmd < xAxis THEN
	servoX_CCW := TRUE;
	servoX_CW := FALSE;
ELSE
	servoX_CCW := FALSE;
	servoX_CW := FALSE;
END_IF
	
IF vYAxisCmd < yAxis THEN
	servoY_CCW := TRUE;
	servoY_CW := FALSE;
ELSIF vYAxisCmd > yAxis THEN
	servoY_CCW := FALSE;
	servoY_CW := TRUE;
ELSE
	servoY_CCW := FALSE;
	servoY_CW := FALSE;
END_IF

	
                  
END_FUNCTION_BLOCK

CONFIGURATION SoftPLC
  RESOURCE Application ON PLC
    {attribute 'qualified_only'}
    VAR_GLOBAL  (* gIO *)
      Garden1_ServoX_CW : BOOL;  (* DO: Garden 1 servo X clock wise turn command *)
      Garden1_ServoX_CCW : BOOL;  (* DO: Garden 1 servo X counter clock wise turn command *)
      Garden1_ServoY_CW : BOOL;  (* DO: Garden 1 servo Y clock wise turn command *)
      Garden1_ServoY_CCW : BOOL;  (* DO: Garden 1 servo Y counter clock wise turn command *)
      Garden1_WaterTankOpenCmd : BOOL;  (* DO: Garden 1 water valve open command *)
      Garden2_ServoX_CW : BOOL;  (* DO: Garden 2 servo X clock wise turn command *)
      Garden2_ServoX_CCW : BOOL;  (* DO: Garden 2 servo X counter clock wise turn command *)
      Garden2_ServoY_CW : BOOL;  (* DO: Garden 2 servo Y clock wise turn command *)
      Garden2_ServoY_CCW : BOOL;  (* DO: Garden 2 servo Y counter clock wise turn command *)
      Garden2_WaterTankOpenCmd : BOOL;  (* DO: Garden 2 water valve open command *)
      Garden3_ServoX_CW : BOOL;  (* DO: Garden 3 servo X clock wise turn command *)
      Garden3_ServoX_CCW : BOOL;  (* DO: Garden 3 servo X counter clock wise turn command *)
      Garden3_ServoY_CW : BOOL;  (* DO: Garden 3 servo Y clock wise turn command *)
      Garden3_ServoY_CCW : BOOL;  (* DO: Garden 3 servo Y counter clock wise turn command *)
      Garden3_WaterTankOpenCmd : BOOL;  (* DO: Garden 3 water valve open command *)
      Garden4_ServoX_CW : BOOL;  (* DO: Garden 4 servo X clock wise turn command *)
      Garden4_ServoX_CCW : BOOL;  (* DO: Garden 4 servo X counter clock wise turn command *)
      Garden4_ServoY_CW : BOOL;  (* DO: Garden 4 servo Y clock wise turn command *)
      Garden4_ServoY_CCW : BOOL;  (* DO: Garden 4 servo Y counter clock wise turn command *)
      Garden4_WaterTankOpenCmd : BOOL;  (* DO: Garden 4 water valve open command *)
      Garden1_ServoX_Offset : INT;  (* AI: Garden 1 servo X offset from starting position *)
      Garden1_ServoY_Offset : INT;  (* AI: Garden 1 servo Y offset from starting position *)
      Garden2_ServoX_Offset : INT;  (* AI: Garden 2 servo X offset from starting position *)
      Garden2_ServoY_Offset : INT;  (* AI: Garden 2 servo Y offset from starting position *)
      Garden3_ServoX_Offset : INT;  (* AI: Garden 3 servo X offset from starting position *)
      Garden3_ServoY_Offset : INT;  (* AI: Garden 3 servo Y offset from starting position *)
      Garden4_ServoX_Offset : INT;  (* AI: Garden 4 servo X offset from starting position *)
      Garden4_ServoY_Offset : INT;  (* AI: Garden 4 servo Y offset from starting position *)
      Garden1_HMI : HMI_Cmds_typ;  (* DI: Garden 1 HMI commands to main program *)
      Garden2_HMI : HMI_Cmds_typ;  (* DI: Garden 2 HMI commands to main program *)
      Garden3_HMI : HMI_Cmds_typ;  (* DI: Garden 3 HMI commands to main program *)
      Garden4_HMI : HMI_Cmds_typ;  (* DI: Garden 4 HMI commands to main program *)
    END_VAR
    TASK VISU_TASK(INTERVAL := T#100ms, PRIORITY := 31);
    TASK Task(INTERVAL := T#20ms, PRIORITY := 1);
    PROGRAM VisuElems.Visu_Prg WITH VISU_TASK : VisuElems.Visu_Prg;
    PROGRAM simu WITH Task : simu;
    PROGRAM main WITH Task : main;
  END_RESOURCE
END_CONFIGURATION
